// TIA Portal V19 export
DATA_BLOCK "RollformerLubr_PERS"   // DB155
// stored: MemoryReserve 100
   VAR RETAIN
      Pump : "LubrMotor_Par";
      Valves1 : Struct
         Control : "LubrValve_Pers";
         Enable_V : Array[1.."ROLL_LUBR_MAXVALVE"] of Bool;
      END_STRUCT;
      Valves2 : Struct
         Control : "LubrValve_Pers";
         Enable_V : Array[1.."ROLL_LUBR_MAXVALVE"] of Bool;
      END_STRUCT;
      Valves3 : Struct
         Control : "LubrValve_Pers";
         Enable_V : Array[1.."ROLL_LUBR_MAXVALVE"] of Bool;
      END_STRUCT;
   END_VAR
BEGIN
   Pump.EnableCheckRotation := FALSE;
   Pump.LowLevelCheckTime := T#3S;
   Pump.RotationFbkCheckTime := T#0MS;
   Valves1.Control.Par.SystemOn := TRUE;
   Valves1.Control.Par.EnableCheckFdbk := FALSE;
   Valves1.Control.Par.CycleFdbkCheckTime := T#0MS;
   Valves1.Control.Par.WorkTime := T#0MS;
   Valves1.Control.Par.ValveONTime := T#1S;
   Valves1.Control.Par.ValveOFFTime := T#1S;
   Valves1.Control.Par.ValvePumpSetPoint := 5;
   Valves1.Control.Par.LubrReqSetPoint := 200.0;
   Valves1.Control.ValvePumpCounter := 0;
   Valves1.Control.LubrReqCounter := 0.0;
   Valves1.Enable_V[1..6] := TRUE;
   Valves2.Control.Par.SystemOn := TRUE;
   Valves2.Control.Par.EnableCheckFdbk := FALSE;
   Valves2.Control.Par.CycleFdbkCheckTime := T#0MS;
   Valves2.Control.Par.WorkTime := T#0MS;
   Valves2.Control.Par.ValveONTime := T#1S;
   Valves2.Control.Par.ValveOFFTime := T#1S;
   Valves2.Control.Par.ValvePumpSetPoint := 2;
   Valves2.Control.Par.LubrReqSetPoint := 200.0;
   Valves2.Control.ValvePumpCounter := 0;
   Valves2.Control.LubrReqCounter := 1777.8497900001;
   Valves2.Enable_V[1..6] := TRUE;
   Valves3.Control.Par.SystemOn := TRUE;
   Valves3.Control.Par.EnableCheckFdbk := FALSE;
   Valves3.Control.Par.CycleFdbkCheckTime := T#0MS;
   Valves3.Control.Par.WorkTime := T#0MS;
   Valves3.Control.Par.ValveONTime := T#1S;
   Valves3.Control.Par.ValveOFFTime := T#1S;
   Valves3.Control.Par.ValvePumpSetPoint := 2;
   Valves3.Control.Par.LubrReqSetPoint := 200.0;
   Valves3.Control.ValvePumpCounter := 0;
   Valves3.Control.LubrReqCounter := 1775.90383600009;
   Valves3.Enable_V[1..6] := TRUE;
END_DATA_BLOCK
